PROGRAM prgComLynus
VAR
	fbCom			: FB_MqttCommunicator_V2;
END_VAR

fbCom(
	bConnect:= TRUE, 
	sUserName:= '806b5b3a-69a5-452f-af78-4b065bd4b761', 
	sUserPassword:= 'fbc367e6-1894-4e5e-8737-325595087c51', 
	strAuthKey := 'TSG88376368072',
	eSavePositionCertificate:= eSavePositionOnPLC.ePostionHardDisk, 
	bConnected=> , 
	bError=> , 
	hrErrorCode=> , 
	eConnectionState=> , 
	eErrorMessage_Out=> );

END_PROGRAM

(* stored: Version 1.1.0.1, ProductVersion 3.1.4024.11
   POU prgComLynus: Id {64c3386a-a78c-459d-aa5f-2c9876969cae}, SpecialFunc None *)
